Universal Robots PolyScope program: al_progs.urp

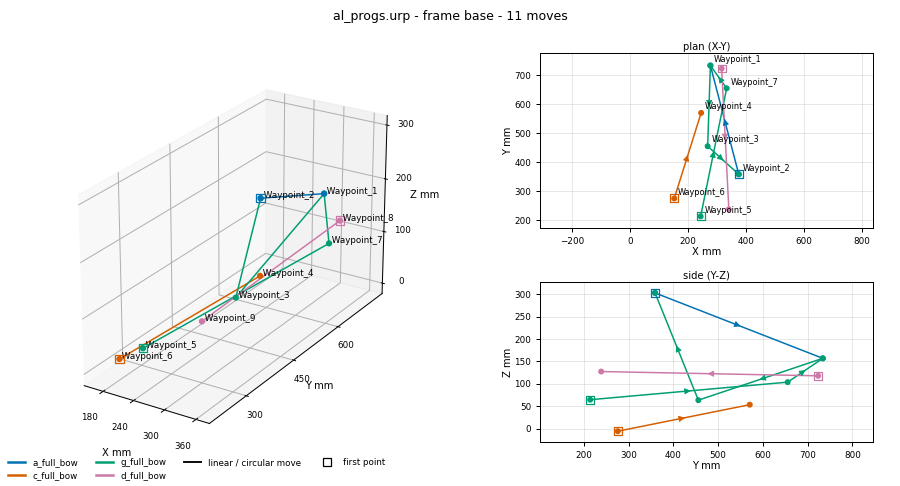
[picture p0: tool path of al_progs.urp in frame base, 11 of 38 moves have a stored position in this frame; points joined in program order, loops and branches not executed]
Program al_progs (installation=string_planes directory=/programs createdIn=5.17.3 lastSavedIn=5.17.3 robotSerialNumber=20245501435)
Calibrated DH parameters: a=[0.000154, -0.137004, -0.385524, -0.00002, 0.000092, 0]; d=[0.162441, 211.794786, -230.585024, 18.923638, 0.099786, 0.09951]; alpha=[1.569493, -0.001902, 0.003874, 1.570111, -1.570167, 0]; deltaTheta=[0, -1.242934, 1.056292, 0.186646, 0.000002, 0.000001]
InitVariablesNode
Robot Program (runOnlyOnce=false)
  string := 1
  note_dur := 1
  bow_dir := 1
  Call a_full_bow
  Call c_full_bow
  Call g_full_bow
  Call d_full_bow
  Call a_to_d
  Call a_to_g
  Call c_to_d
  Call d_to_a
  Call d_to_g
  Call d_to_c
  Call g_to_a
  Call g_to_c
  Call g_to_d
SubProgram -> g_to_d
SubProgram -> g_to_c
SubProgram -> g_to_a
SubProgram -> d_to_c
SubProgram -> d_to_g
SubProgram -> d_to_a
SubProgram -> c_to_d
SubProgram -> a_to_g
SubProgram -> a_to_d
SubProgram -> d_full_bow
SubProgram -> g_full_bow
SubProgram -> c_full_bow
SubProgram -> a_full_bow
SubProgram a_full_bow (keepSynchronizedWithDisk=false) programFile=/programs/a_full_bow.urp
  bow_dir := True
  note_dur := 3
  Timer (action=Start) variable(name=timer_1)
  If bow_dir
    MoveL speed 250 mm/s, acceleration 1200 mm/s^2 (useActiveTCP=true) feature=Base
      Waypoint Waypoint_2: TCP in base x=374.969 y=359.127 z=303.035 mm, rx=1.6275 ry=2.3373 rz=-1.1146 rad; joints [-156.117, -66.368, 101.552, -88.734, -114.429, -168.118] deg; TCP offset x=28.21 y=-96.107 z=-99.69 mm, rx=0 ry=0 rz=0 rad
        Until EXPRESSION (allowActions=false) ExpressionBranch=timer_1≟note_dur
  Else 
    MoveL speed 250 mm/s, acceleration 1200 mm/s^2 (useActiveTCP=true) feature=Base
      Waypoint Waypoint_1: TCP in base x=277.237 y=734.032 z=156.892 mm, rx=1.7389 ry=2.3104 rz=-1.1078 rad; joints [-126.647, -28.123, 54.729, -74.616, -91.964, -141.812] deg; TCP offset x=28.21 y=-96.107 z=-99.69 mm, rx=0 ry=0 rz=0 rad
        Until EXPRESSION (allowActions=false) ExpressionBranch=timer_1≟note_dur
  SuppressedNode
    MoveL speed 250 mm/s, acceleration 1200 mm/s^2 (useActiveTCP=true) feature=Base
      Waypoint Waypoint_1: TCP in base x=277.237 y=734.032 z=156.892 mm, rx=1.7389 ry=2.3104 rz=-1.1078 rad; joints [-126.647, -28.123, 54.729, -74.616, -91.964, -141.812] deg
      Waypoint Waypoint_3: motionParameters(blendRadius=0.05); TCP in base x=335.809 y=527.638 z=230.762 mm, rx=1.7389 ry=2.3104 rz=-1.1078 rad; joints [-141.244, -51.172, 87.867, -86.053, -101.589, -152.842] deg; TCP offset x=28.21 y=-96.107 z=-99.69 mm, rx=0 ry=0 rz=0 rad
      Waypoint Waypoint_2: TCP in base x=393.128 y=325.659 z=303.053 mm, rx=1.7389 ry=2.3104 rz=-1.1078 rad; joints [-160.523, -67.347, 103.242, -90.17, -113.569, -168.748] deg
  Timer (action=Stop) variable=timer_1
  Timer (action=Reset) variable=timer_1
SubProgram c_full_bow (keepSynchronizedWithDisk=false) programFile=/programs/c_full_bow.urp
  bow_dir := True
  note_dur := 1
  Timer (action=Start) variable(name=timer_2)
  If bow_dir≟ True
    MoveL speed 250 mm/s, acceleration 1200 mm/s^2 (useActiveTCP=true) feature=Base
      Waypoint Waypoint_6: TCP in base x=152.636 y=275.824 z=-5.984 mm, rx=-1.6122 ry=-1.6008 rz=0.7404 rad; joints [-153.501, -26.653, 138.52, -151.348, -62.645, -165.795] deg
        Until EXPRESSION (allowActions=false) ExpressionBranch=timer_1≟note_dur
  Else 
    MoveL speed 250 mm/s, acceleration 1200 mm/s^2 (useActiveTCP=true) feature=Base
      Waypoint Waypoint_4: TCP in base x=245.284 y=570.71 z=53.266 mm, rx=-1.8425 ry=-1.3918 rz=0.0687 rad; joints [-132.226, -24.798, 96.314, -169.322, -42.692, -112.607] deg
        Until EXPRESSION (allowActions=false) ExpressionBranch=timer_1≟note_dur
  SuppressedNode
    MoveL speed 250 mm/s, acceleration 1200 mm/s^2 (useActiveTCP=true) feature=Base
      Waypoint Waypoint_4: TCP in base x=245.284 y=570.71 z=53.266 mm, rx=-1.8425 ry=-1.3918 rz=0.0687 rad; joints [-132.226, -24.798, 96.314, -169.322, -42.692, -112.607] deg
      Waypoint Waypoint_1: TCP in base x=195.249 y=411.456 z=21.268 mm, rx=-1.7342 ry=-1.5169 rz=0.4322 rad; joints [-140.231, -30.936, 122.536, -154.99, -45.802, -143.197] deg
      Waypoint Waypoint_6: TCP in base x=152.636 y=275.824 z=-5.984 mm, rx=-1.6122 ry=-1.6008 rz=0.7404 rad; joints [-153.501, -26.653, 138.52, -151.348, -62.645, -165.795] deg
  Timer (action=Stop) variable=timer_2
  Timer (action=Reset) variable=timer_2
SubProgram g_full_bow (keepSynchronizedWithDisk=false) programFile=/programs/g_full_bow.urp
  bow_dir := True
  note_dur := 1
  Timer (action=Start) variable(name=timer_3)
  If bow_dir
    MoveL speed 250 mm/s, acceleration 1200 mm/s^2 (useActiveTCP=true) feature=Base
      Waypoint Waypoint_5: TCP in base x=243.61 y=214.062 z=64.413 mm, rx=-1.5874 ry=-1.9212 rz=0.9621 rad; joints [-169.308, -44.602, 138.126, -133.88, -94.42, -177.775] deg
        Until EXPRESSION (allowActions=false) ExpressionBranch=timer_1≟note_dur
  Else 
    MoveL speed 250 mm/s, acceleration 1200 mm/s^2 (useActiveTCP=true) feature=Base
      Waypoint Waypoint_7: TCP in base x=333.313 y=655.49 z=103.651 mm, rx=-1.6491 ry=-1.7982 rz=0.6657 rad; joints [-132.463, -27.757, 71.844, -100.482, -56.044, -147.729] deg
        Until EXPRESSION (allowActions=false) ExpressionBranch=timer_1≟note_dur
  MoveL speed 250 mm/s, acceleration 1200 mm/s^2 (useActiveTCP=true) feature=Base
    Waypoint Waypoint_1: TCP in base x=277.237 y=734.032 z=156.892 mm, rx=1.7389 ry=2.3104 rz=-1.1078 rad; joints [-126.647, -28.123, 54.729, -74.616, -91.964, -141.812] deg; TCP offset x=28.21 y=-96.107 z=-99.69 mm, rx=0 ry=0 rz=0 rad
    Waypoint Waypoint_3: motionParameters(blendRadius=0.05); TCP in base x=267.763 y=455.808 z=63.345 mm, rx=-1.6064 ry=-1.9107 rz=0.8702 rad; joints [-141.616, -39.193, 108.914, -115.288, -70.782, -159.12] deg; TCP offset x=28.21 y=-96.107 z=-99.69 mm, rx=0 ry=0 rz=0 rad
    Waypoint Waypoint_2: TCP in base x=374.969 y=359.127 z=303.035 mm, rx=1.6275 ry=2.3373 rz=-1.1146 rad; joints [-156.117, -66.368, 101.552, -88.734, -114.429, -168.118] deg
  Timer (action=Stop) variable=timer_3
  Timer (action=Reset) variable=timer_3
SubProgram d_full_bow (keepSynchronizedWithDisk=false) programFile=/programs/d_full_bow.urp
  bow_dir := True
  note_dur := 1
  Timer (action=Start) variable(name=timer_4)
  If bow_dir≟ False
    MoveL speed 250 mm/s, acceleration 1200 mm/s^2 (useActiveTCP=true) feature=Base
      Waypoint Waypoint_8: TCP in base x=316.077 y=723.624 z=117.8 mm, rx=-1.5349 ry=-2.2386 rz=1.1274 rad; joints [-128.458, -21.868, 50.818, -72.931, -81.953, -152.853] deg
        Until EXPRESSION (allowActions=false) ExpressionBranch=timer_1≟note_dur
  Else 
    MoveL speed 250 mm/s, acceleration 1200 mm/s^2 (useActiveTCP=true) feature=Base
      Waypoint Waypoint_9: TCP in base x=340.806 y=238.625 z=127.338 mm, rx=-1.5375 ry=-2.1223 rz=1.0863 rad; joints [-167.854, -53.469, 123.568, -113.681, -104.543, -179.466] deg
        Until EXPRESSION (allowActions=false) ExpressionBranch=timer_1≟note_dur
  SuppressedNode
    MoveL speed 250 mm/s, acceleration 1200 mm/s^2 (useActiveTCP=true) feature=Base
      Waypoint Waypoint_1: TCP in base x=331.973 y=720.894 z=108.291 mm, rx=-1.645 ry=-2.1081 rz=1.0591 rad; joints [-129.773, -21.651, 52.373, -76.468, -76.907, -149.022] deg
      Waypoint Waypoint_2: motionParameters(blendRadius=0.05); TCP in base x=332.259 y=481.199 z=108.291 mm, rx=-1.645 ry=-2.1081 rz=1.0591 rad; joints [-144.031, -41.816, 97.865, -100.392, -86.961, -159.136] deg
      Waypoint Waypoint_3: TCP in base x=332.566 y=223.853 z=108.291 mm, rx=-1.645 ry=-2.1081 rz=1.0591 rad; joints [-170.229, -51.627, 126.122, -120.942, -105.516, -177.767] deg
  Timer (action=Stop) variable=timer_4
  Timer (action=Reset) variable=timer_4
SubProgram a_to_d (keepSynchronizedWithDisk=false) programFile=/programs/string_crossings/a_to_d.urp
  bow_section := -1
  If bow_section≟-1
    MoveJ speed 60 deg/s, acceleration 80 deg/s^2 (useActiveTCP=true) feature=Base
      Waypoint Waypoint_10 (Relative): relativeFromPosition TCP in base x=277.235 y=734.032 z=156.893 mm, rx=1.7389 ry=2.3104 rz=-1.1077 rad; joints [-126.647, -28.124, 54.729, -74.617, -91.964, -141.812] deg; TCP in base x=316.092 y=723.606 z=117.8 mm, rx=-1.5349 ry=-2.2386 rz=1.1274 rad; joints [-128.46, -21.869, 50.821, -72.931, -81.953, -152.855] deg
  ElseIf bow_section≟0
    MoveJ speed 60 deg/s, acceleration 80 deg/s^2 (useActiveTCP=true) feature=Base
      Waypoint Waypoint_11 (Relative): relativeFromPosition TCP in base x=327.074 y=542.849 z=231.417 mm, rx=1.6821 ry=2.3247 rz=-1.1115 rad; joints [-139.55, -50.207, 85.865, -84.66, -102.289, -153.001] deg; TCP in base x=329.632 y=457.693 z=123.027 mm, rx=-1.5368 ry=-2.1747 rz=1.1049 rad; joints [-145.135, -44.399, 100.427, -98.676, -90.572, -164.15] deg
  Else 
    MoveJ speed 60 deg/s, acceleration 80 deg/s^2 (useActiveTCP=true) feature=Base
      Waypoint Waypoint_12 (Relative): relativeFromPosition TCP in base x=374.965 y=359.133 z=303.036 mm, rx=1.6274 ry=2.3373 rz=-1.1146 rad; joints [-156.116, -66.368, 101.551, -88.734, -114.43, -168.118] deg; TCP in base x=340.8 y=238.63 z=127.345 mm, rx=-1.5375 ry=-2.1223 rz=1.0863 rad; joints [-167.853, -53.47, 123.568, -113.68, -104.544, -179.466] deg
SubProgram a_to_g (keepSynchronizedWithDisk=false) programFile=/programs/string_crossings/a_to_g.urp
  bow_section := -1
  If bow_section≟-1
    MoveJ speed 60 deg/s, acceleration 80 deg/s^2 (useActiveTCP=true) feature=Base
      Waypoint Waypoint_13 (Relative): relativeFromPosition TCP in base x=277.254 y=734.024 z=156.891 mm, rx=1.739 ry=2.3104 rz=-1.1077 rad; joints [-126.649, -28.124, 54.73, -74.617, -91.964, -141.812] deg; TCP in base x=333.304 y=655.498 z=103.667 mm, rx=-1.6491 ry=-1.7982 rz=0.6657 rad; joints [-132.463, -27.758, 71.844, -100.482, -56.045, -147.728] deg
  ElseIf bow_section≟0
    MoveJ speed 60 deg/s, acceleration 80 deg/s^2 (useActiveTCP=true) feature=Base
      Waypoint Waypoint_14 (Relative): relativeFromPosition TCP in base x=327.375 y=541.709 z=231.859 mm, rx=1.6817 ry=2.3248 rz=-1.1115 rad; joints [-139.64, -50.32, 85.997, -84.694, -102.36, -153.081] deg; TCP in base x=267.746 y=455.84 z=63.354 mm, rx=-1.6064 ry=-1.9108 rz=0.8701 rad; joints [-141.612, -39.193, 108.911, -115.29, -70.78, -159.12] deg
  Else 
    MoveJ speed 60 deg/s, acceleration 80 deg/s^2 (useActiveTCP=true) feature=Base
      Waypoint Waypoint_15 (Relative): relativeFromPosition TCP in base x=374.965 y=359.139 z=303.04 mm, rx=1.6275 ry=2.3374 rz=-1.1145 rad; joints [-156.115, -66.368, 101.551, -88.734, -114.428, -168.118] deg; TCP in base x=243.614 y=214.06 z=64.414 mm, rx=-1.5873 ry=-1.9212 rz=0.9621 rad; joints [-169.308, -44.603, 138.126, -133.881, -94.42, -177.776] deg
SubProgram c_to_d (keepSynchronizedWithDisk=false) programFile=/programs/string_crossings/c_to_d.urp
  bow_section := -1
  If bow_section≟-1
    MoveJ speed 60 deg/s, acceleration 80 deg/s^2 (useActiveTCP=true) feature=Base
      Waypoint Waypoint_16 (Relative): relativeFromPosition TCP in base x=245.287 y=570.708 z=53.279 mm, rx=-1.8425 ry=-1.3918 rz=0.0687 rad; joints [-132.226, -24.799, 96.314, -169.323, -42.69, -112.608] deg; TCP in base x=316.071 y=723.616 z=117.783 mm, rx=-1.5349 ry=-2.2386 rz=1.1275 rad; joints [-128.458, -21.868, 50.821, -72.931, -81.953, -152.853] deg
  ElseIf bow_section≟0
    MoveJ speed 60 deg/s, acceleration 80 deg/s^2 (useActiveTCP=true) feature=Base
      Waypoint Waypoint_17 (Relative): relativeFromPosition TCP in base x=195.299 y=411.479 z=21.277 mm, rx=-1.7342 ry=-1.517 rz=0.432 rad; joints [-140.233, -30.937, 122.528, -154.99, -45.802, -143.198] deg; TCP in base x=337.286 y=452.569 z=146.265 mm, rx=-1.6084 ry=-2.1978 rz=1.0429 rad; joints [-146.229, -47.168, 100.749, -99.804, -91.441, -163.024] deg
  Else 
    MoveJ speed 60 deg/s, acceleration 80 deg/s^2 (useActiveTCP=true) feature=Base
      Waypoint Waypoint_18 (Relative): relativeFromPosition TCP in base x=152.636 y=275.828 z=-5.99 mm, rx=-1.6121 ry=-1.6008 rz=0.7404 rad; joints [-153.501, -26.652, 138.519, -151.349, -62.643, -165.795] deg; TCP in base x=340.805 y=238.622 z=127.329 mm, rx=-1.5375 ry=-2.1223 rz=1.0863 rad; joints [-167.854, -53.467, 123.568, -113.681, -104.544, -179.467] deg
SubProgram d_to_a (keepSynchronizedWithDisk=false) programFile=/programs/string_crossings/d_to_a.urp
  bow_section := 1
  If bow_section≟-1
    MoveJ speed 60 deg/s, acceleration 80 deg/s^2 (useActiveTCP=true) feature=Base
      Waypoint Waypoint_19 (Relative): relativeFromPosition TCP in base x=316.068 y=723.618 z=117.805 mm, rx=-1.5349 ry=-2.2387 rz=1.1274 rad; joints [-128.458, -21.869, 50.821, -72.933, -81.954, -152.854] deg; TCP in base x=277.256 y=734.024 z=156.889 mm, rx=1.7389 ry=2.3104 rz=-1.1078 rad; joints [-126.649, -28.123, 54.728, -74.617, -91.964, -141.814] deg
  ElseIf bow_section≟0
    MoveJ speed 60 deg/s, acceleration 80 deg/s^2 (useActiveTCP=true) feature=Base
      Waypoint Waypoint_20 (Relative): relativeFromPosition TCP in base x=329.63 y=457.702 z=123.03 mm, rx=-1.5368 ry=-2.1747 rz=1.1049 rad; joints [-145.135, -44.399, 100.427, -98.676, -90.57, -164.149] deg; TCP in base x=327.082 y=542.85 z=231.412 mm, rx=1.6821 ry=2.3247 rz=-1.1115 rad; joints [-139.551, -50.206, 85.865, -84.66, -102.288, -153.001] deg
  Else 
    MoveJ speed 60 deg/s, acceleration 80 deg/s^2 (useActiveTCP=true) feature=Base
      Waypoint Waypoint_21 (Relative): relativeFromPosition TCP in base x=340.803 y=238.631 z=127.342 mm, rx=-1.5375 ry=-2.1223 rz=1.0863 rad; joints [-167.853, -53.469, 123.568, -113.681, -104.544, -179.465] deg; TCP in base x=374.961 y=359.138 z=303.027 mm, rx=1.6274 ry=2.3373 rz=-1.1146 rad; joints [-156.115, -66.367, 101.552, -88.732, -114.429, -168.117] deg
SubProgram d_to_g (keepSynchronizedWithDisk=false) programFile=/programs/string_crossings/d_to_g.urp
  bow_section := -1
  If bow_section≟-1
    MoveJ speed 60 deg/s, acceleration 80 deg/s^2 (useActiveTCP=true) feature=Base
      Waypoint Waypoint_22 (Relative): relativeFromPosition TCP in base x=316.1 y=723.608 z=117.809 mm, rx=-1.5349 ry=-2.2386 rz=1.1274 rad; joints [-128.46, -21.869, 50.82, -72.931, -81.953, -152.853] deg; TCP in base x=333.322 y=655.489 z=103.666 mm, rx=-1.649 ry=-1.7982 rz=0.6656 rad; joints [-132.464, -27.757, 71.843, -100.482, -56.044, -147.73] deg
  ElseIf bow_section≟0
    MoveJ speed 60 deg/s, acceleration 80 deg/s^2 (useActiveTCP=true) feature=Base
      Waypoint Waypoint_23 (Relative): relativeFromPosition TCP in base x=329.884 y=452.806 z=123.116 mm, rx=-1.5368 ry=-2.1735 rz=1.1045 rad; joints [-145.541, -44.677, 101.077, -99.034, -90.804, -164.42] deg; TCP in base x=267.754 y=455.821 z=63.355 mm, rx=-1.6064 ry=-1.9107 rz=0.8702 rad; joints [-141.614, -39.194, 108.914, -115.288, -70.781, -159.121] deg
  Else 
    MoveJ speed 60 deg/s, acceleration 80 deg/s^2 (useActiveTCP=true) feature=Base
      Waypoint Waypoint_24 (Relative): relativeFromPosition TCP in base x=340.793 y=238.63 z=127.341 mm, rx=-1.5374 ry=-2.1223 rz=1.0863 rad; joints [-167.853, -53.469, 123.569, -113.681, -104.544, -179.467] deg; TCP in base x=243.611 y=214.066 z=64.414 mm, rx=-1.5873 ry=-1.9212 rz=0.9621 rad; joints [-169.307, -44.603, 138.125, -133.881, -94.42, -177.776] deg
SubProgram d_to_c (keepSynchronizedWithDisk=false) programFile=/programs/string_crossings/d_to_c.urp
  bow_section := -1
  If bow_section≟-1
    MoveJ speed 60 deg/s, acceleration 80 deg/s^2 (useActiveTCP=true) feature=Base
      Waypoint Waypoint_25 (Relative): relativeFromPosition TCP in base x=316.087 y=723.603 z=117.786 mm, rx=-1.5349 ry=-2.2386 rz=1.1275 rad; joints [-128.46, -21.869, 50.823, -72.931, -81.954, -152.853] deg; TCP in base x=245.285 y=570.708 z=53.285 mm, rx=-1.8425 ry=-1.3918 rz=0.0687 rad; joints [-132.226, -24.799, 96.314, -169.323, -42.691, -112.607] deg
  ElseIf bow_section≟0
    MoveJ speed 60 deg/s, acceleration 80 deg/s^2 (useActiveTCP=true) feature=Base
      Waypoint Waypoint_26 (Relative): relativeFromPosition TCP in base x=337.283 y=452.564 z=146.255 mm, rx=-1.6083 ry=-2.1978 rz=1.0429 rad; joints [-146.229, -47.167, 100.75, -99.804, -91.441, -163.026] deg; TCP in base x=195.29 y=411.468 z=21.275 mm, rx=-1.7343 ry=-1.5169 rz=0.4321 rad; joints [-140.233, -30.937, 122.531, -154.99, -45.8, -143.197] deg
  Else 
    MoveJ speed 60 deg/s, acceleration 80 deg/s^2 (useActiveTCP=true) feature=Base
      Waypoint Waypoint_27 (Relative): relativeFromPosition TCP in base x=340.787 y=238.628 z=127.316 mm, rx=-1.5374 ry=-2.1222 rz=1.0864 rad; joints [-167.853, -53.466, 123.57, -113.68, -104.543, -179.467] deg; TCP in base x=152.628 y=275.821 z=-5.995 mm, rx=-1.6121 ry=-1.6008 rz=0.7404 rad; joints [-153.501, -26.651, 138.52, -151.349, -62.642, -165.796] deg
SubProgram g_to_a (keepSynchronizedWithDisk=false) programFile=/programs/string_crossings/g_to_a.urp
  bow_section := -1
  If bow_section≟-1
    MoveJ speed 60 deg/s, acceleration 80 deg/s^2 (useActiveTCP=true) feature=Base
      Waypoint Waypoint_28 (Relative): relativeFromPosition TCP in base x=333.304 y=655.506 z=103.679 mm, rx=-1.6491 ry=-1.7982 rz=0.6657 rad; joints [-132.462, -27.759, 71.843, -100.48, -56.044, -147.727] deg; TCP in base x=277.25 y=734.024 z=156.888 mm, rx=1.739 ry=2.3104 rz=-1.1078 rad; joints [-126.649, -28.124, 54.73, -74.618, -91.963, -141.811] deg
  ElseIf bow_section≟0
    MoveJ speed 60 deg/s, acceleration 80 deg/s^2 (useActiveTCP=true) feature=Base
      Waypoint Waypoint_29 (Relative): relativeFromPosition TCP in base x=267.753 y=455.828 z=63.352 mm, rx=-1.6064 ry=-1.9107 rz=0.8701 rad; joints [-141.613, -39.193, 108.913, -115.288, -70.779, -159.12] deg; TCP in base x=327.364 y=541.729 z=231.867 mm, rx=1.6818 ry=2.3248 rz=-1.1114 rad; joints [-139.638, -50.32, 85.996, -84.695, -102.358, -153.079] deg
  Else 
    MoveJ speed 60 deg/s, acceleration 80 deg/s^2 (useActiveTCP=true) feature=Base
      Waypoint Waypoint_30 (Relative): relativeFromPosition TCP in base x=243.623 y=214.066 z=64.409 mm, rx=-1.5873 ry=-1.9212 rz=0.9621 rad; joints [-169.307, -44.602, 138.124, -133.879, -94.42, -177.776] deg; TCP in base x=374.975 y=359.143 z=303.031 mm, rx=1.6275 ry=2.3373 rz=-1.1145 rad; joints [-156.115, -66.366, 101.55, -88.735, -114.429, -168.117] deg
SubProgram g_to_c (keepSynchronizedWithDisk=false) programFile=/programs/string_crossings/g_to_c.urp
  bow_section := -1
  If bow_section≟-1
    MoveJ speed 60 deg/s, acceleration 80 deg/s^2 (useActiveTCP=true) feature=Base
      Waypoint Waypoint_31 (Relative): relativeFromPosition TCP in base x=333.313 y=655.493 z=103.664 mm, rx=-1.6491 ry=-1.7981 rz=0.6657 rad; joints [-132.463, -27.758, 71.844, -100.481, -56.042, -147.727] deg; TCP in base x=245.295 y=570.7 z=53.28 mm, rx=-1.8424 ry=-1.3918 rz=0.0687 rad; joints [-132.227, -24.799, 96.314, -169.321, -42.687, -112.61] deg
  ElseIf bow_section≟0
    MoveJ speed 60 deg/s, acceleration 80 deg/s^2 (useActiveTCP=true) feature=Base
      Waypoint Waypoint_32 (Relative): relativeFromPosition TCP in base x=267.761 y=455.827 z=63.349 mm, rx=-1.6064 ry=-1.9107 rz=0.8701 rad; joints [-141.614, -39.193, 108.912, -115.289, -70.779, -159.12] deg; TCP in base x=195.266 y=411.465 z=21.275 mm, rx=-1.7342 ry=-1.5169 rz=0.4321 rad; joints [-140.231, -30.937, 122.534, -154.989, -45.801, -143.196] deg
  Else 
    MoveJ speed 60 deg/s, acceleration 80 deg/s^2 (useActiveTCP=true) feature=Base
      Waypoint Waypoint_33 (Relative): relativeFromPosition TCP in base x=243.617 y=214.085 z=64.401 mm, rx=-1.5874 ry=-1.9213 rz=0.9621 rad; joints [-169.304, -44.6, 138.123, -133.882, -94.42, -177.774] deg; TCP in base x=152.648 y=275.83 z=-5.999 mm, rx=-1.6122 ry=-1.6008 rz=0.7404 rad; joints [-153.502, -26.651, 138.518, -151.349, -62.642, -165.794] deg
SubProgram g_to_d (keepSynchronizedWithDisk=false) programFile=/programs/string_crossings/g_to_d.urp
  bow_section := -1
  If bow_section≟-1
    MoveJ speed 60 deg/s, acceleration 80 deg/s^2 (useActiveTCP=true) feature=Base
      Waypoint Waypoint_34 (Relative): relativeFromPosition TCP in base x=333.345 y=655.475 z=103.654 mm, rx=-1.6491 ry=-1.7982 rz=0.6656 rad; joints [-132.466, -27.757, 71.843, -100.482, -56.044, -147.73] deg; TCP in base x=316.098 y=723.605 z=117.805 mm, rx=-1.5349 ry=-2.2386 rz=1.1275 rad; joints [-128.46, -21.869, 50.821, -72.93, -81.955, -152.853] deg
  ElseIf bow_section≟0
    MoveJ speed 60 deg/s, acceleration 80 deg/s^2 (useActiveTCP=true) feature=Base
      Waypoint Waypoint_35 (Relative): relativeFromPosition TCP in base x=267.758 y=455.827 z=63.35 mm, rx=-1.6064 ry=-1.9107 rz=0.8702 rad; joints [-141.614, -39.193, 108.913, -115.288, -70.78, -159.119] deg; TCP in base x=337.277 y=452.587 z=146.27 mm, rx=-1.6083 ry=-2.1978 rz=1.0429 rad; joints [-146.227, -47.168, 100.748, -99.801, -91.438, -163.024] deg
  Else 
    MoveJ speed 60 deg/s, acceleration 80 deg/s^2 (useActiveTCP=true) feature=Base
      Waypoint Waypoint_36 (Relative): relativeFromPosition TCP in base x=243.623 y=214.066 z=64.413 mm, rx=-1.5874 ry=-1.9212 rz=0.962 rad; joints [-169.308, -44.603, 138.124, -133.881, -94.42, -177.776] deg; TCP in base x=340.792 y=238.623 z=127.333 mm, rx=-1.5375 ry=-2.1223 rz=1.0864 rad; joints [-167.854, -53.469, 123.57, -113.681, -104.544, -179.466] deg
